// TIA Portal V20 export
VAR_GLOBAL   // PLC tag table "06_ProductionData"
END_VAR
VAR_GLOBAL CONSTANT   // user constants
   NO_DATASETS_CYCLETIMER : Int := 8;   // SICAR: Anzahl Datensätze Taktzeiten / SICAR: Number of data sets Cycle Timer
   NO_DATASETS_LIMITVALUES : Int := 2;   // SICAR: Anzahl Datensätze Grenzwerte / SICAR: Number of data sets Limit Value
   NO_DATASETS_SHIFTCOUNTER : Int := 2;   // SICAR: Anzahl Datensätze Schichtzähler / SICAR: Number of data sets Shift Counter
   NO_DATASETS_COUNTER : Int := 2;   // SICAR: Anzahl Datensätze Zähler / SICAR: Number of data sets Counter
END_VAR
